(* CODESYS project MachineSimulation.project

Project tree, tasks and I/O mapping:
  Device : CODESYS Control Win V3, 3S - Smart Software Solutions GmbH, order no. 305021, version 3.5.11.30
    application Application
      libraries: Standard, * (System)
      MachineSimulation/
        task MainTask (cyclic, interval t#20ms, priority 1) calls PLC_PRG
      task VISU_TASK (cyclic, interval 100 ms, priority 31) calls VisuElems.Visu_Prg
      program PLC_PRG [ST]
      global variables GVL_Modbus
      visualisation MachineVisualization
      image pool Background
    Ethernet : Ethernet, Eaton Automation, version 3.5.11.0
        settings: IPAddress = [192,168,1,100]; SubnetMask = [255,255,255,0]; GatewayAddress = [0,0,0,0]; MACAddress = [16#00,16#0C,16#29,16#78,16#27,16#A6]; NetworkInterfaceName = 'Ethernet0'; NetworkInterfaceName = "Ethernet0"; SaveCommunicationSettings = FALSE
      ModbusTCP_Slave_Device : ModbusTCP Slave Device, 3S - Smart Software Solutions GmbH, version 3.5.11.0
          settings: Unit-ID = 1
          output Application.GVL_Modbus.MB_MachineRunning : WORD  // Outputs.Outputs
          output Application.GVL_Modbus.MB_AlarmActive : WORD  // Outputs.Outputs
          output Application.GVL_Modbus.MB_ProductionCount : WORD  // Outputs.Outputs
          output Application.GVL_Modbus.MB_Temperature_x10 : WORD  // Outputs.Outputs
          unmapped channels: Inputs, Outputs
  libraries: VisuSymbols, 3.5.10.0 (System)
  text list GlobalTextList
*)

// Device/Application/GVL_Modbus
{attribute 'qualified_only'}
VAR_GLOBAL
	
	// Registradores enviados ao cliente Modbus
	
    MB_MachineRunning : WORD := 0;
    MB_AlarmActive : WORD := 0;
    MB_ProductionCount : WORD := 0;
    MB_Temperature_x10 : WORD := 0;
	
	// Variaveis globais
	
    StartCommand : BOOL := FALSE;
    StopCommand : BOOL := FALSE;
    ResetProductionCommand : BOOL := FALSE;

    MachineRunning : BOOL := FALSE;
    AlarmActive : BOOL := FALSE;

    ProductionCount : INT := 0;
    Temperature : REAL := 25.0;
END_VAR

// Device/Application/PLC_PRG
PROGRAM PLC_PRG
VAR
	// Temporizadores locais da simulação
    ProductionTimer : TON;
    TemperatureTimer : TON;
END_VAR

// =====================================================
// Controle de partida
// =====================================================

IF GVL_Modbus.StartCommand AND NOT GVL_Modbus.AlarmActive THEN
    GVL_Modbus.MachineRunning := TRUE;
    GVL_Modbus.StartCommand := FALSE;
END_IF;

// =====================================================
// Controle de parada
// =====================================================

IF GVL_Modbus.StopCommand THEN
    GVL_Modbus.MachineRunning := FALSE;
    GVL_Modbus.StopCommand := FALSE;
END_IF;

// =====================================================
// Reset do contador de produção
// =====================================================

IF GVL_Modbus.ResetProductionCommand THEN
    GVL_Modbus.ProductionCount := 0;
    GVL_Modbus.ResetProductionCommand := FALSE;
END_IF;

// =====================================================
// Simulação da produção
// Uma peça é produzida a cada 2 segundos
// =====================================================

ProductionTimer(
    IN := GVL_Modbus.MachineRunning AND NOT ProductionTimer.Q,
    PT := T#2S
);

IF ProductionTimer.Q THEN
    GVL_Modbus.ProductionCount := GVL_Modbus.ProductionCount + 1;
END_IF;

// =====================================================
// Atualização periódica da temperatura
// =====================================================

TemperatureTimer(
    IN := NOT TemperatureTimer.Q,
    PT := T#1S
);

IF TemperatureTimer.Q THEN

    IF GVL_Modbus.MachineRunning THEN
        GVL_Modbus.Temperature := GVL_Modbus.Temperature + 1.0;
    ELSE
        GVL_Modbus.Temperature := GVL_Modbus.Temperature - 0.5;
    END_IF;

END_IF;

// =====================================================
// Limite mínimo da temperatura
// =====================================================

IF GVL_Modbus.Temperature < 25.0 THEN
    GVL_Modbus.Temperature := 25.0;
END_IF;

// =====================================================
// Alarme e parada por temperatura
// =====================================================

IF GVL_Modbus.Temperature >= 45.0 THEN
    GVL_Modbus.AlarmActive := TRUE;
    GVL_Modbus.MachineRunning := FALSE;

ELSIF GVL_Modbus.Temperature <= 40.0 THEN
    GVL_Modbus.AlarmActive := FALSE;
END_IF;

// =====================================================
// Atualização dos registradores de saída Modbus
// =====================================================

IF GVL_Modbus.MachineRunning THEN
    GVL_Modbus.MB_MachineRunning := 1;
ELSE
    GVL_Modbus.MB_MachineRunning := 0;
END_IF;

IF GVL_Modbus.AlarmActive THEN
    GVL_Modbus.MB_AlarmActive := 1;
ELSE
    GVL_Modbus.MB_AlarmActive := 0;
END_IF;

GVL_Modbus.MB_ProductionCount :=
    INT_TO_WORD(GVL_Modbus.ProductionCount);

GVL_Modbus.MB_Temperature_x10 :=
    REAL_TO_WORD(GVL_Modbus.Temperature * 10.0);

END_PROGRAM

// Device/Application/MachineVisualization
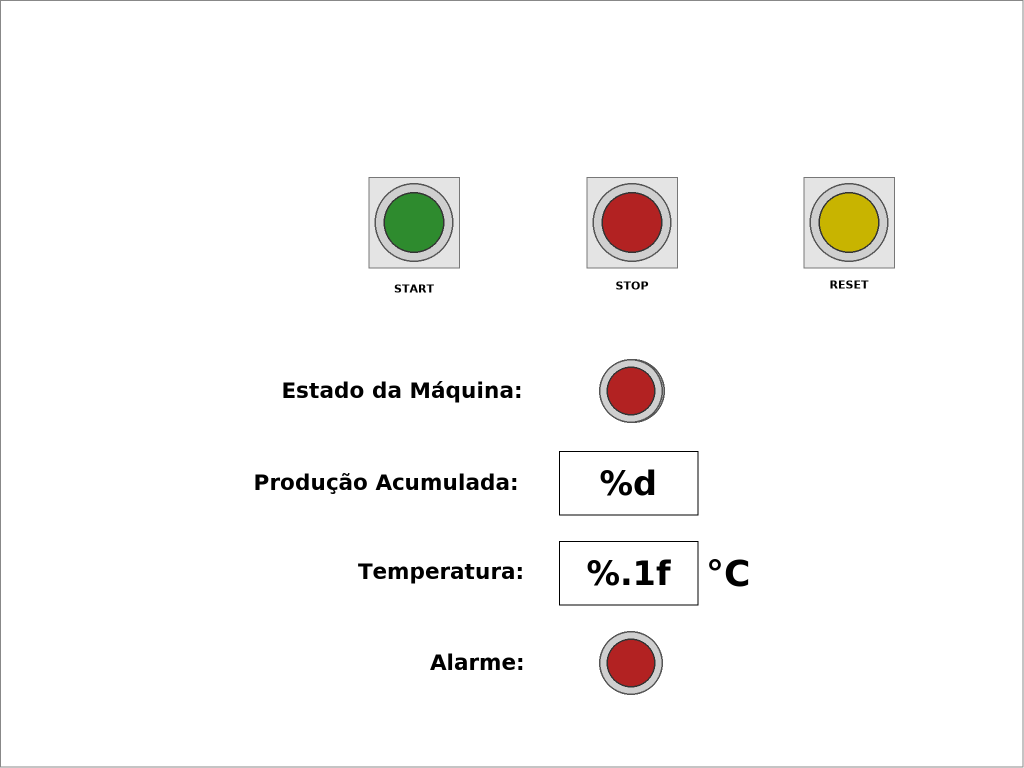
VISUALIZATION MachineVisualization  // 1024x768, background image ec433c39-f5a7-4105-9918-ba6c92bd6da5
    PushSwitch (366,177 96x91), variable: GVL_Modbus.StartCommand, behaviour: TAP, style: Switch-PushSwitch-Green
    PushSwitch (584,177 96x91), variable: GVL_Modbus.StopCommand, behaviour: TAP, style: Switch-PushSwitch-Red
    PushSwitch (801,177 96x91), variable: GVL_Modbus.ResetProductionCommand, behaviour: TAP, style: Switch-PushSwitch-Yellow
    Label (339,274 150x30), "START"
    Label (557,271 150x30), "STOP"
    Label (774,270 150x30), "RESET"
    Label (270,365 264x51), "Estado da Máquina:"
    Label (238,457 296x51), "Produção Acumulada:"
    Label (348,546 186x51), "Temperatura:"
    Label (421,637 113x51), "Alarme:"
    Lamp1 (592,354 82x74), variable: GVL_Modbus.MachineRunning, invisible if: GVL_Modbus.StopCommand, style: Lamp-Lamp1-Green
    Lamp1 (590,354 82x74), variable: GVL_Modbus.StopCommand, invisible if: GVL_Modbus.MachineRunning, style: Lamp-Lamp1-Red
    Rectangle (559,451 139x64), "%d", text variable: GVL_Modbus.ProductionCount
    Rectangle (559,541 139x64), "%.1f", text variable: GVL_Modbus.Temperature
    Lamp1 (590,626 82x74), variable: GVL_Modbus.AlarmActive, invisible if: GVL_Modbus.MachineRunning, style: Lamp-Lamp1-Red
    Label (698,545 61x57), "°C"
END_VISUALIZATION
